// Mitsubishi GX Works2 project: 检测肥料12.18   PLC: FX3U/FX3UC

PROGRAM MAIN
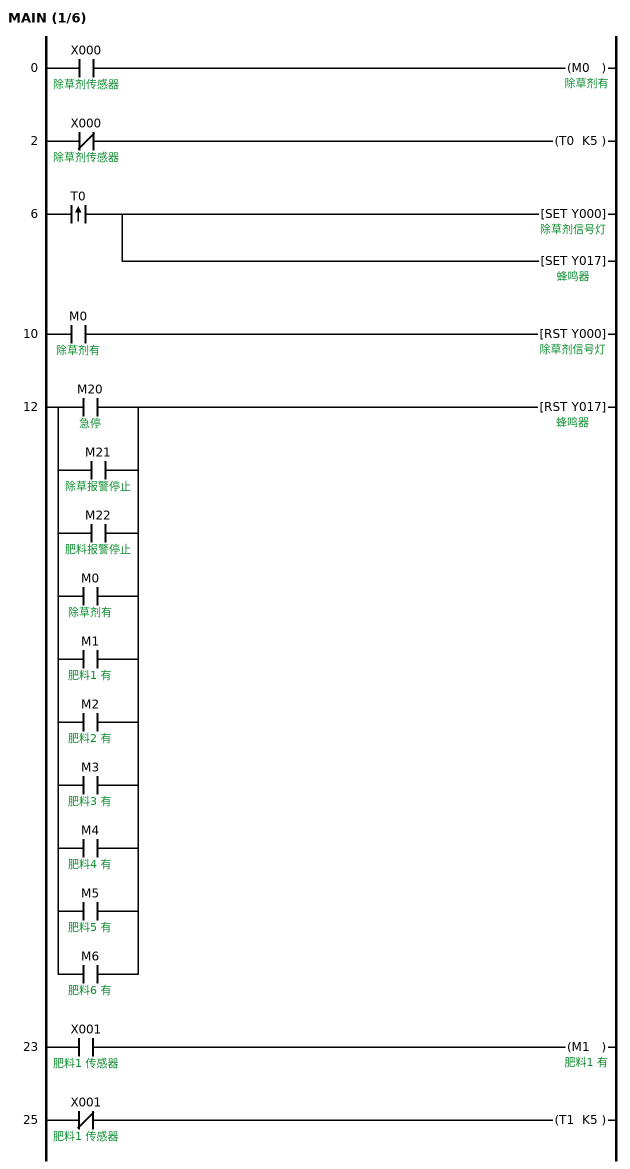
0     LD      X000  ; 除草剂传感器
      OUT     M0  ; 除草剂有
2     LDI     X000  ; 除草剂传感器
      OUT     T0 K5
6     LDP     T0
      SET     Y000  ; 除草剂信号灯
      SET     Y017  ; 蜂鸣器
10    LD      M0  ; 除草剂有
      RST     Y000  ; 除草剂信号灯
12    LD      M20  ; 急停
      OR      M21  ; 除草报警停止
      OR      M22  ; 肥料报警停止
      OR      M0  ; 除草剂有
      OR      M1  ; 肥料1 有
      OR      M2  ; 肥料2 有
      OR      M3  ; 肥料3 有
      OR      M4  ; 肥料4 有
      OR      M5  ; 肥料5 有
      OR      M6  ; 肥料6 有
      RST     Y017  ; 蜂鸣器
23    LD      X001  ; 肥料1 传感器
      OUT     M1  ; 肥料1 有
25    LDI     X001  ; 肥料1 传感器
      OUT     T1 K5
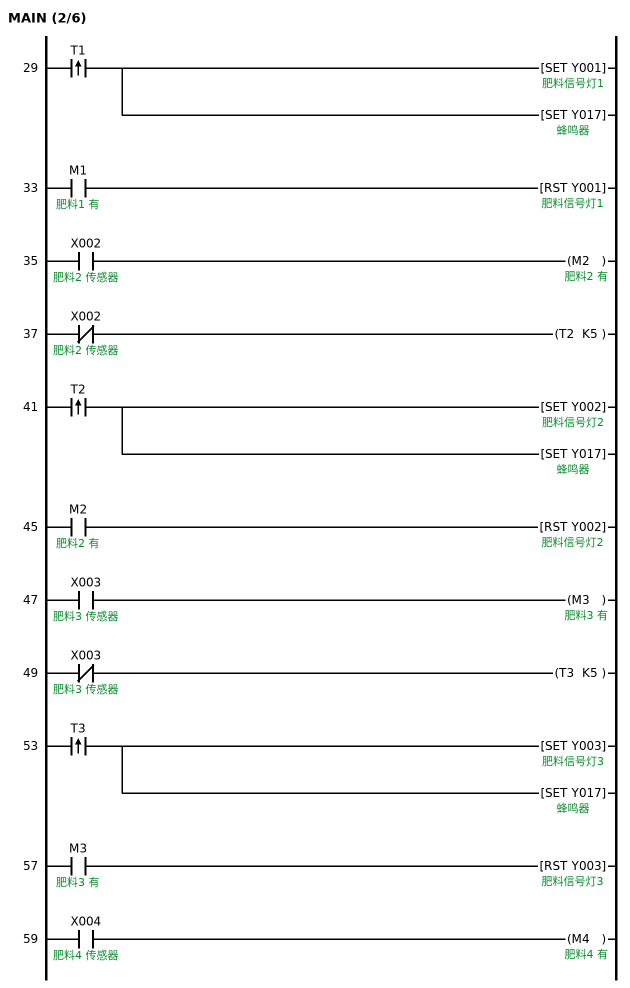
29    LDP     T1
      SET     Y001  ; 肥料信号灯1
      SET     Y017  ; 蜂鸣器
33    LD      M1  ; 肥料1 有
      RST     Y001  ; 肥料信号灯1
35    LD      X002  ; 肥料2 传感器
      OUT     M2  ; 肥料2 有
37    LDI     X002  ; 肥料2 传感器
      OUT     T2 K5
41    LDP     T2
      SET     Y002  ; 肥料信号灯2
      SET     Y017  ; 蜂鸣器
45    LD      M2  ; 肥料2 有
      RST     Y002  ; 肥料信号灯2
47    LD      X003  ; 肥料3 传感器
      OUT     M3  ; 肥料3 有
49    LDI     X003  ; 肥料3 传感器
      OUT     T3 K5
53    LDP     T3
      SET     Y003  ; 肥料信号灯3
      SET     Y017  ; 蜂鸣器
57    LD      M3  ; 肥料3 有
      RST     Y003  ; 肥料信号灯3
59    LD      X004  ; 肥料4 传感器
      OUT     M4  ; 肥料4 有
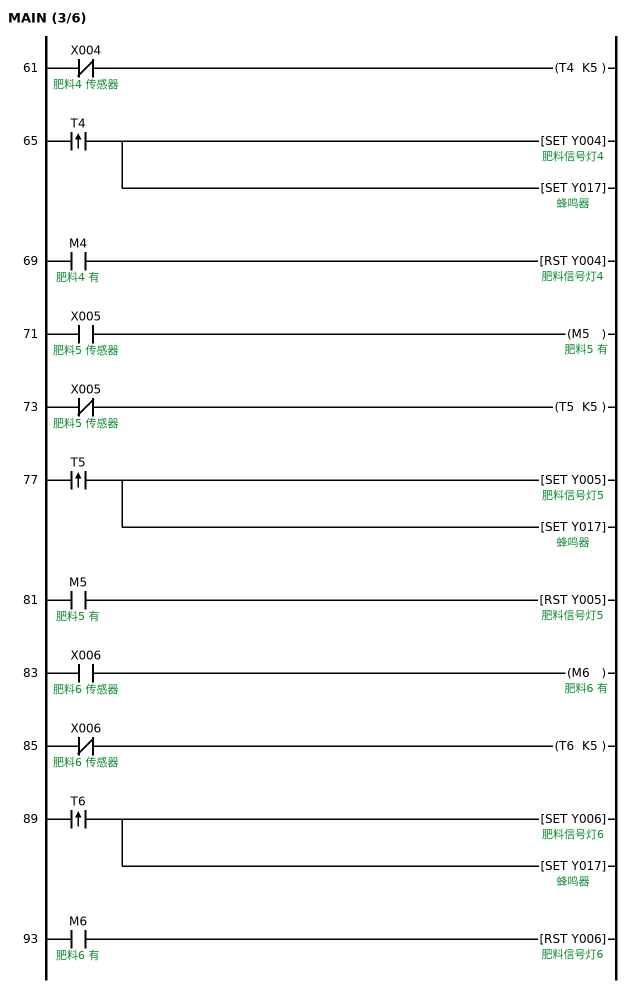
61    LDI     X004  ; 肥料4 传感器
      OUT     T4 K5
65    LDP     T4
      SET     Y004  ; 肥料信号灯4
      SET     Y017  ; 蜂鸣器
69    LD      M4  ; 肥料4 有
      RST     Y004  ; 肥料信号灯4
71    LD      X005  ; 肥料5 传感器
      OUT     M5  ; 肥料5 有
73    LDI     X005  ; 肥料5 传感器
      OUT     T5 K5
77    LDP     T5
      SET     Y005  ; 肥料信号灯5
      SET     Y017  ; 蜂鸣器
81    LD      M5  ; 肥料5 有
      RST     Y005  ; 肥料信号灯5
83    LD      X006  ; 肥料6 传感器
      OUT     M6  ; 肥料6 有
85    LDI     X006  ; 肥料6 传感器
      OUT     T6 K5
89    LDP     T6
      SET     Y006  ; 肥料信号灯6
      SET     Y017  ; 蜂鸣器
93    LD      M6  ; 肥料6 有
      RST     Y006  ; 肥料信号灯6
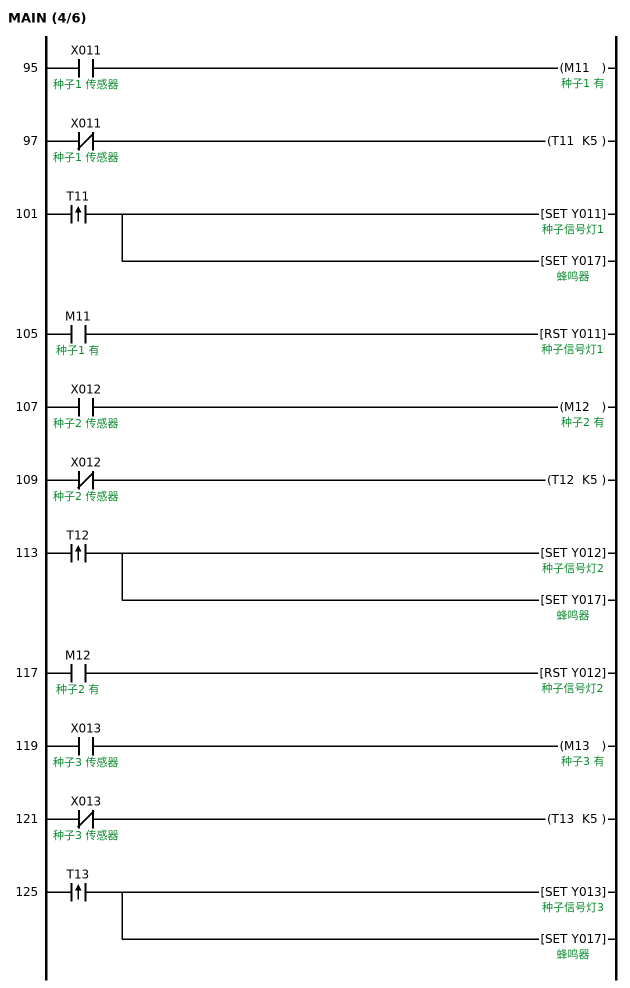
95    LD      X011  ; 种子1 传感器
      OUT     M11  ; 种子1 有
97    LDI     X011  ; 种子1 传感器
      OUT     T11 K5
101   LDP     T11
      SET     Y011  ; 种子信号灯1
      SET     Y017  ; 蜂鸣器
105   LD      M11  ; 种子1 有
      RST     Y011  ; 种子信号灯1
107   LD      X012  ; 种子2 传感器
      OUT     M12  ; 种子2 有
109   LDI     X012  ; 种子2 传感器
      OUT     T12 K5
113   LDP     T12
      SET     Y012  ; 种子信号灯2
      SET     Y017  ; 蜂鸣器
117   LD      M12  ; 种子2 有
      RST     Y012  ; 种子信号灯2
119   LD      X013  ; 种子3 传感器
      OUT     M13  ; 种子3 有
121   LDI     X013  ; 种子3 传感器
      OUT     T13 K5
125   LDP     T13
      SET     Y013  ; 种子信号灯3
      SET     Y017  ; 蜂鸣器
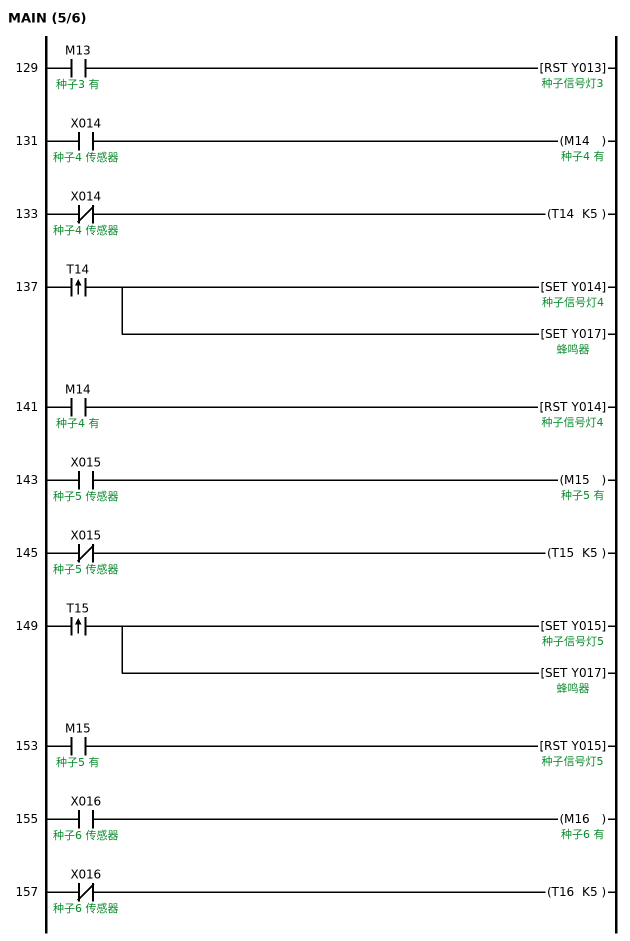
129   LD      M13  ; 种子3 有
      RST     Y013  ; 种子信号灯3
131   LD      X014  ; 种子4 传感器
      OUT     M14  ; 种子4 有
133   LDI     X014  ; 种子4 传感器
      OUT     T14 K5
137   LDP     T14
      SET     Y014  ; 种子信号灯4
      SET     Y017  ; 蜂鸣器
141   LD      M14  ; 种子4 有
      RST     Y014  ; 种子信号灯4
143   LD      X015  ; 种子5 传感器
      OUT     M15  ; 种子5 有
145   LDI     X015  ; 种子5 传感器
      OUT     T15 K5
149   LDP     T15
      SET     Y015  ; 种子信号灯5
      SET     Y017  ; 蜂鸣器
153   LD      M15  ; 种子5 有
      RST     Y015  ; 种子信号灯5
155   LD      X016  ; 种子6 传感器
      OUT     M16  ; 种子6 有
157   LDI     X016  ; 种子6 传感器
      OUT     T16 K5
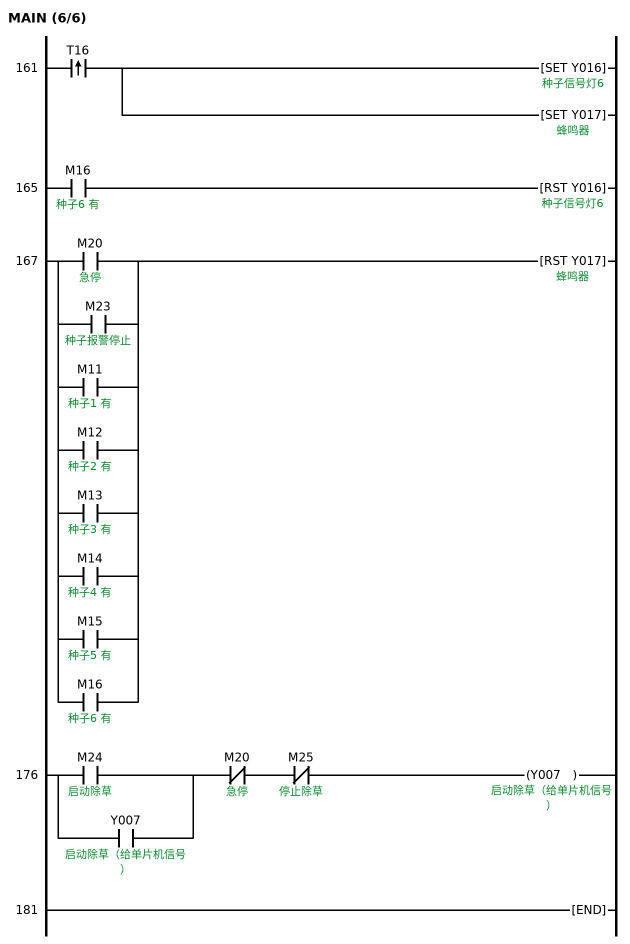
161   LDP     T16
      SET     Y016  ; 种子信号灯6
      SET     Y017  ; 蜂鸣器
165   LD      M16  ; 种子6 有
      RST     Y016  ; 种子信号灯6
167   LD      M20  ; 急停
      OR      M23  ; 种子报警停止
      OR      M11  ; 种子1 有
      OR      M12  ; 种子2 有
      OR      M13  ; 种子3 有
      OR      M14  ; 种子4 有
      OR      M15  ; 种子5 有
      OR      M16  ; 种子6 有
      RST     Y017  ; 蜂鸣器
176   LD      M24  ; 启动除草
      OR      Y007  ; 启动除草（给单片机信号）
      ANI     M20  ; 急停
      ANI     M25  ; 停止除草
      OUT     Y007  ; 启动除草（给单片机信号）
181   END
END_PROGRAM

// device comments not shown above
Y010  ; 蜂鸣器
M7  ; 肥料7 有
